FUNCTION ASCF_GetVDIntOutputList : Word
VAR_INPUT
	Index		: INT;
END_VAR

VAR_OUTPUT
	QC			: BYTE;
	Value		: DINT;
END_VAR

VAR_IN_OUT
	OutputList	: ARRAY[*] OF ASCF_CL_OutputType;		//Output-Element of the Adaptive Logic.
END_VAR

VAR
	tempLowerBound	: DINT;
	tempUpperBound	: DINT;
	tempResult		: WORD;
	tempUnionType	: ASCF_UnionType;				//Union type that holds only one of its possible data types at a time. The type can be selected via the "Typeselector". Independent of the selected type, every value has a quality code "VQC".
	constErrors		: ASCF_CL_EnumErrors;				//Enumeration type of the error codes of the Adaptive Logic.
	constUnionTypes	: ASCF_EnumUnionTypes;			//Enumeration type of the valid values for the "Typeselector" of a "GVR_unionType"-UDT.
END_VAR



tempResult := ASCF_GetValueOutputList(Index := Index, Value => tempUnionType, OutputList := OutputList);

IF tempResult <> constErrors.None THEN
    ASCF_GetVDIntOutputList := tempResult;
    RETURN;
END_IF;

IF tempUnionType.Typeselector <> constUnionTypes.VDINT THEN
    ASCF_GetVDIntOutputList := constErrors.TypesDoNotMatch;
    RETURN;
END_IF;

QC := tempUnionType.VQC;
Value := tempUnionType.VDINT;
ASCF_GetVDIntOutputList := constErrors.None;

END_FUNCTION

(* stored: Version 1.1.0.1, ProductVersion 3.1.4026.4
   POU ASCF_GetVDIntOutputList: Id {46f9b208-b9bd-4fdf-95f2-cc689a80edde}, SpecialFunc None *)
